// TIA Portal V16 export
// export: Created 2024-09-05T15:58:41.8073085Z, ExportSetting WithDefaults, DisplayName Totally Integrated Automation Portal, DisplayVersion V16 Update 6, DisplayName TIA Portal Version Control Interface, DisplayVersion V16 Update 2, DisplayName TIA Portal Openness, DisplayVersion V16 Update 6, DisplayName STEP 7 Professional, DisplayVersion V16 Update 6, DisplayName STEP 7 Safety, DisplayVersion V16, DisplayName WinCC Advanced, DisplayVersion V16 Update 6
VAR_GLOBAL   // PLC tag table "plc"
   iAirPressure AT %I0.1 : Bool;
   iEmergencyStopHydraulics1 AT %I1.0 : Bool;
   iEmergencyStopHydraulics2 AT %I1.1 : Bool;
   iBtnOpenServiceDoors1 AT %I1.2 : Bool;
   iBtnResetServiceDoors1 AT %I1.3 : Bool;
   iBtnOpenServiceDoors2 AT %I1.4 : Bool;
   iBtnResetServiceDoors2 AT %I1.5 : Bool;
   qServiceDoorUnlock1 AT %Q1.0 : Bool;
   qServiceDoorUnlock2 AT %Q1.1 : Bool;
   qLighthouseRed AT %Q1.3 : Bool;
   qLighthouseOrange AT %Q1.4 : Bool;
   qLighthouseGreen AT %Q1.6 : Bool;
   qLighthouseWhite AT %Q1.7 : Bool;
   qLEDDoors1Open AT %Q3.0 : Bool;
   qLEDDoors2Open AT %Q3.1 : Bool;
   qLEDDoors1EMG AT %Q3.3 : Bool;
   qLEDDoors2EMG AT %Q3.4 : Bool;
   iAntennaStartCycle AT %I0.0 : Bool;
   qMS6reset AT %Q3.6 : Bool;
   qResetServiceDoors AT %Q0.1 : Bool;
   qSafetyScannerReset AT %Q0.2 : Bool;
   qLEDsafetyScannerReset AT %Q1.2 : Bool;
   iSafetyScannerResetNotRequired AT %I2.7 : Bool;
   iServiceDoorClosed1 AT %I1.6 : Bool;
   iServiceDoorClosed2 AT %I1.7 : Bool;
   qAudioSignal AT %Q0.0 : Bool;
   qLighthouseBlue AT %Q1.5 : Bool;
   iEmergencyStopConveyor AT %I2.3 : Bool;
END_VAR
